TYPE Roller_y :
STRUCT
	roller	: Roller;
	photo_sensor	: ARRAY[0..1] OF BOOL;
END_STRUCT
END_TYPE

(* stored: Version 1.1.0.1, ProductVersion 3.1.4024.12
   DUT Roller_y: Id {6db26d65-57da-4e29-9f6a-51e4f57cecc8} *)
